RoboDK station: Custom_Assistive_UR5e.rdk

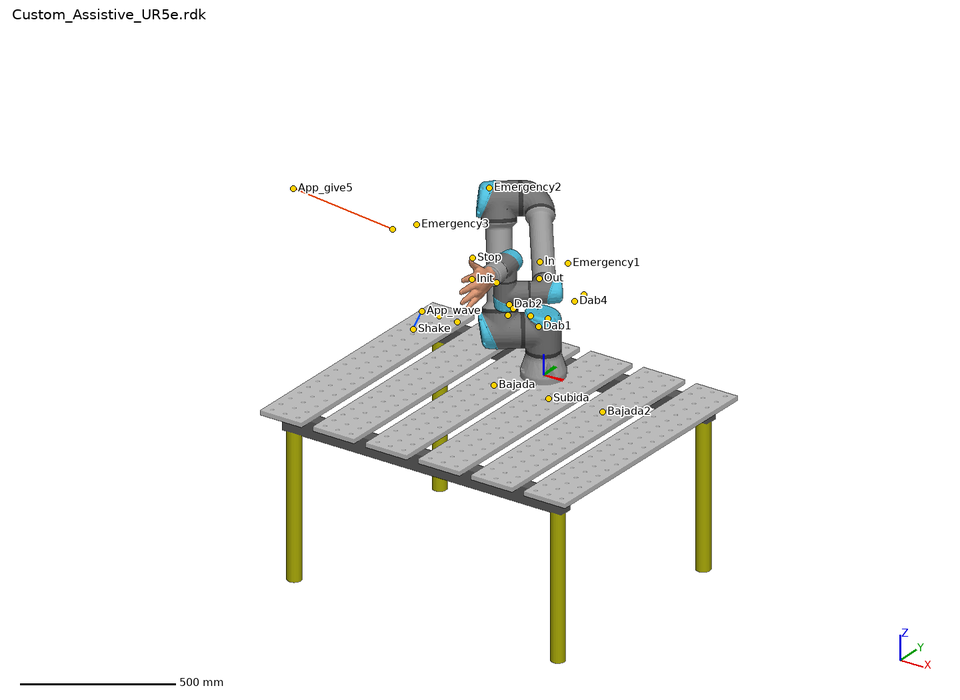
[picture v0: the station drawn from its stored meshes, robots at their saved joint values, targets as dots, program paths as lines]
Station Assistive_UR5e_SW (saved by RoboDK 5.9.2). Poses are relative to the parent item; angles as X-Y-Z fixed-axis rotations.
  - frame UR5e Base at (0, 0, 0) mm, rotated rx 0 ry 0 rz 5.71 deg
    - robot UR5e: 6 axes, payload 5 kg, reach 850 mm, repeatability 0.03 mm, weight 18.4 kg
        modified DH rows (alpha deg, a mm, theta deg, d mm): 0, 0, 0, 162.5; 90, 0, 180, 0; 0, 425, 0, 0; 0, 392.25, 0, 133.3; -90, 0, 0, 99.7; 90, 0, 180, 99.6
        joint limits [-360, -360, -360, -360, -360, -360] to [360, 360, 360, 360, 360, 360]; home [0, -90, -90, 0, 90, 0]; saved at [-57.836, -69.983, -134.335, -335.683, -302.164, 180]
      - tool Hand, TCP at (0, 0, 50) mm, size 54.8 x 155.9 x 193.5 mm, geometry from Hand.stl
  - frame World at (0, 0, 0) mm
    - object Table at (0, 0, 0) mm, size 1193.8 x 965.2 x 609.6 mm, geometry from welding_table.sld
    - target Init (Cartesian target) at (0, -400, 500) mm, rotated rx 90 ry 0 rz 0 deg; joints [-57.836, -85.391, -107.167, 172.559, -57.836, 0] of UR5e
    - target App_wave (Cartesian target) at (0, -680, 500) mm, rotated rx 90 ry 0 rz 0 deg; joints [75.444, 18.986, -92.472, -106.514, -75.444, 180] of UR5e
    - target Wave (Cartesian target) at (67.6, -676.63, 500) mm, rotated rx -120.53 ry -80.83 rz -46.18 deg; joints [-91.174, -132.208, -29.443, -171.146, -190.197, 124.748] of UR5e
    - target Bajada (Cartesian target) at (266.61, -656.75, 300) mm, rotated rx 168.48 ry -36.56 rz 9.52 deg; joints [-68.848, -118.561, -85.504, -41.08, -240.155, 207.874] of UR5e
    - target Subida (Cartesian target) at (465.62, -636.87, 300) mm, rotated rx 15.33 ry -52.65 rz 170.3 deg; joints [-57.574, -135.775, -73.382, 265.429, -135.289, -234.622] of UR5e
    - target Bajada2 (Cartesian target) at (664.63, -616.98, 300) mm, rotated rx 158.97 ry -63.45 rz 21.58 deg; joints [-45.449, -150.106, -44.369, -15.769, 124.078, -118.259] of UR5e
    - target Dab1 (Cartesian target) at (362.2, -543.84, 491.58) mm, rotated rx 114.89 ry -7.59 rz 96.22 deg; joints [-61.176, -108.98, -82.438, 323.837, 145.591, 146.277] of UR5e
    - target Dab2 (Cartesian target) at (172.25, -436.94, 472.75) mm, rotated rx -88.95 ry 1.72 rz 87.14 deg; joints [106.123, -65.2, 92.171, 155.534, 155.259, 3.997] of UR5e
    - target Dab3 (Cartesian target) at (328.74, -444.84, 469.88) mm, rotated rx 2.86 ry 2.34 rz 84.31 deg; joints [-46.283, -131.145, -73.523, 113.656, 93.55, 214.795] of UR5e
    - target Dab4 (Cartesian target) at (401.61, -399.53, 535.21) mm, rotated rx 71.1 ry 7.22 rz 94.57 deg; joints [-47.929, -112.144, -91.526, -308.852, -224.153, 192.834] of UR5e
    - target Dab5 (Cartesian target) at (-37.15, -427.6, 349.98) mm, rotated rx -36.77 ry -72.63 rz 17.8 deg; joints [-68.138, -109.309, -93.931, -175.141, -310.685, 112.825] of UR5e
    - target Stop (Cartesian target) at (104.87, -544.1, 663.71) mm, rotated rx 0.91 ry -1.55 rz 86.03 deg; joints [-70.892, -185.036, 93.55, -180.311, -90.055, 61.225] of UR5e
    - target Go1 (Cartesian target) at (316.63, -648.89, 561.79) mm, rotated rx 49.4 ry 19.98 rz -49.73 deg; joints [-49.459, -113.761, -74.832, -94.483, -38.889, -98.973] of UR5e
    - target Go2 (Cartesian target) at (379.57, -614.2, 561.79) mm, rotated rx 58.49 ry 33.17 rz -24.02 deg; joints [-44.044, -110.239, -68.401, -139.477, -40.944, -71.589] of UR5e
    - target Go3 (Cartesian target) at (416.76, -366.91, 549.07) mm, rotated rx 47.88 ry -15.82 rz -54.02 deg; joints [-24.969, -113.592, -91.387, -23.416, -59.658, -129.459] of UR5e
    - target Emergency1 (Cartesian target) at (369.19, -390.07, 657.09) mm, rotated rx 44.43 ry 11.41 rz 90.31 deg; joints [-47.177, -173.069, 88.339, -216.71, 235.13, -332.996] of UR5e
    - target Emergency2 (Cartesian target) at (61.72, -390.13, 839.8) mm, rotated rx 0.28 ry -2.71 rz 88.94 deg; joints [-66.54, -75.224, -86.77, -110.493, -88.878, 59.804] of UR5e
    - target Emergency3 (Cartesian target) at (-184.47, -444.32, 661.33) mm, rotated rx -51.27 ry -2.69 rz 104.32 deg; joints [-87.083, -77.116, -101.742, -100.832, -39.343, 99.003] of UR5e
    - target RCP_up (Cartesian target) at (81.09, -375.96, 501.44) mm, rotated rx -128.4 ry -76.75 rz -107.76 deg; joints [-64.734, -68.392, -102.25, -197.556, -93.584, 99.936] of UR5e
    - target RCP_down (Cartesian target) at (122.59, -344.82, 409.26) mm, rotated rx -128.4 ry -76.75 rz -102.05 deg; joints [-54.283, -64.026, -118.214, -185.943, -88.888, 100.612] of UR5e
    - target Out (Cartesian target) at (172.95, -269.64, 500) mm, rotated rx 90 ry 10.97 rz -41 deg; joints [-10.547, -75.277, -100.9, 176.177, 36.16, -10.97] of UR5e
    - target In (Cartesian target) at (125.44, -199.1, 517.45) mm, rotated rx 90 ry 10.97 rz -35.3 deg; joints [10.571, -61.614, -106.506, 168.121, 51.572, -10.97] of UR5e
    - target Shake (joint target) at (-300, -300, 200) mm, rotated rx 90 ry 0 rz 0 deg; joints [-129.97, -95.332, -131.473, -133.195, -129.97, 0] of UR5e
    - target Give5 (joint target) at (-380.86, -300, 533.82) mm, rotated rx 0 ry 0 rz 90 deg; joints [-125.814, -94.091, -116.939, 301.03, -90, 125.814] of UR5e
    - target App_give5 (joint target) at (-810.86, -238.62, 533.82) mm, rotated rx 0 ry 0 rz 90 deg; joints [-154.528, -143.977, -40.15, 274.127, -90, 154.528] of UR5e
    - target Wave2 (Cartesian target) at (0, -680, 500) mm, rotated rx 165.29 ry 0 rz 86.57 deg; joints [-81.878, -163.91, 50.211, -153.291, 104.409, 101.932] of UR5e
  - program Init (3 instructions, listed below)
  - program Hand_shake (5 instructions, listed below)
  - program Give_me_5! (5 instructions, listed below)
  - program MainProgram (4 instructions, listed below)
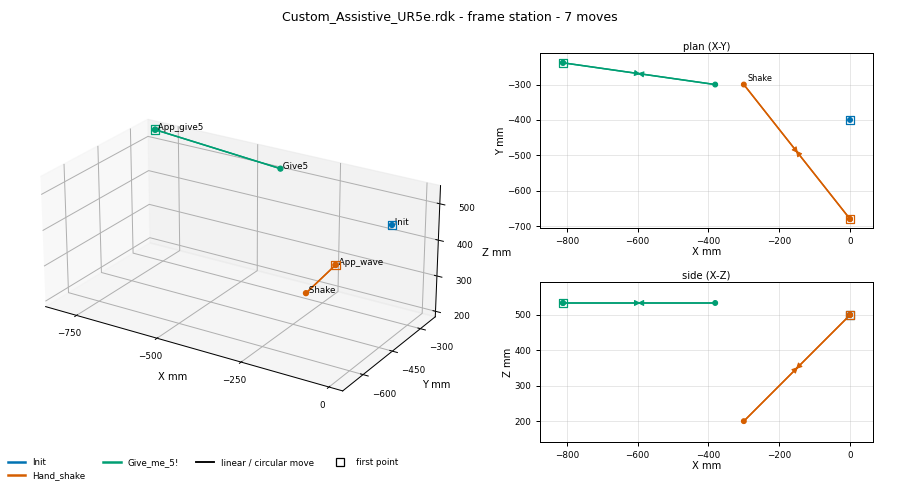
[picture p0: tool path of Custom_Assistive_UR5e.rdk in frame station, 7 of 7 moves have a stored position in this frame; points joined in program order, loops and branches not executed]

--- program Init (robot UR5e) ---
  Est. Ref.: UR5e Base
  Est. herr: Hand
  MoveJ (Init)

--- program Hand_shake (robot UR5e) ---
  Est. Ref.: UR5e Base
  Est. herr: Hand
  MoveL (App_shake) -> target App_wave
  MoveL (Shake)
  MoveL (App_shake) -> target App_wave

--- program Give_me_5! (robot UR5e) ---
  Est. Ref.: UR5e Base
  Est. herr: Hand
  MoveL (App_give5)
  MoveL (Give5)
  MoveL (App_give5)

--- program MainProgram (robot UR5e) ---
  Llamar Init
  Llamar Hand_shake
  Llamar Give_me_5!
  Llamar Init
